VAR_GLOBAL CONSTANT
	iC_MAX_NUM_LINES_IN_FILE : UINT := 1000;
	iC_MAX_STRING_LENGTH : UINT := 25;
END_VAR

(* stored: Version 1.1.0.1
   GVL GLOBAL_CONSTANTS: Id {5db04770-c9e9-4ac7-b5ab-1ad35faa6d54} *)
